FUNCTION_BLOCK FB_ESPNow
VAR_INPUT
END_VAR
VAR_OUTPUT
END_VAR
VAR
END_VAR

END_FUNCTION_BLOCK

(* stored: Version 1.1.0.1, ProductVersion 3.1.4024.9
   POU FB_ESPNow: Id {8a6cba47-4e1d-444c-964e-af34a8ee43ab}, SpecialFunc None *)
